Fanuc KAREL source: kt00104.KL

-- PROVISIONAL review KL for V1013-1; original PC SHA256 b9d29e7733c5f2ece26c1b25ca90903393618c629f9fe56938f453b449a533a8
-- Incomplete behavior may be omitted. Consult companion uncertainty JSON. Do not deploy.
PROGRAM KT00104
%NOLOCKGROUP
VAR
  I1 : INTEGER
  OUT : REAL
-- UNRESOLVED_DECL H2 type=002017
BEGIN
  -- UNRESOLVED_PC offsets 5-16; opcodes 2E,23
  -- UNRESOLVED_PC offsets 21-35; opcodes 2E,22,9D,33,B4
  -- UNRESOLVED_PC offsets 40-66; opcodes 21,22,9D,33,B3,64,29,64,29,6C,23
  -- UNRESOLVED_PC offsets 71-75; opcodes 7F
END KT00104
